(*
Finds the owning entity of a given component in the Entity-Component system.  
This function may involve a costly search operation, iterating through all components.
Returns:
- `Ok` - Successfully retrieves the `I_Entity` that owns the component.
- `Err.Itf0` - iIn = 0.
- `Err.InvRef` - Invalid output reference.
- `Err.NotFound` - No owning entity is found, returning null.
*)
FUNCTION GetOwnerFromRaw : Result
VAR_INPUT
	iIn: I_RawComponent;
	iOut: REFERENCE TO I_Entity;
END_VAR
VAR
	_iComp		: I_Component;
END_VAR

IF iIn = 0 THEN
	GetOwnerFromRaw := Err.Itf0;
	RETURN;
END_IF

IF NOT __ISVALIDREF(iOut) THEN
	GetOwnerFromRaw := Err.InvRef;
	RETURN;
END_IF

WHILE IsOk(GetNextEntity(iOut)) DO
	WHILE IsOk(iOut.GetNextComp(_iComp)) DO
		IF _iComp.Raw = iIn THEN
			GetOwnerFromRaw := Ok;
			RETURN;
		END_IF
	END_WHILE
END_WHILE

GetOwnerFromRaw := Err.NotFound;

END_FUNCTION

(* stored: Version 1.1.0.1
   POU GetOwnerFromRaw: Id {a3b7220f-6050-4211-8801-8b108ece1681}, SpecialFunc None *)
